RoboDK station: MPC Dental Surgery.rdk

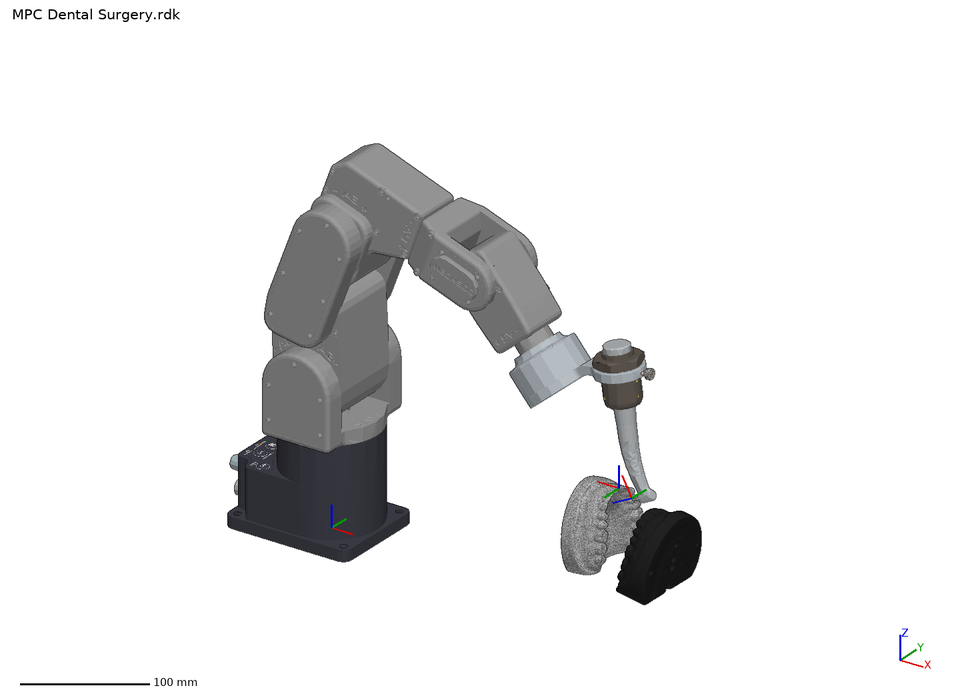
[picture v0: the station drawn from its stored meshes, robots at their saved joint values, targets as dots, program paths as lines]
Station MPC Dental Surgery (saved by RoboDK 5.3.5). Poses are relative to the parent item; angles as X-Y-Z fixed-axis rotations.
  - frame Mecademic Meca500 R3 Base at (0, 0, 0) mm
    - robot Mecademic Meca500 R3: 6 axes, payload 0.5 kg, reach 330 mm, repeatability 0.005 mm, weight 4.5 kg
        modified DH rows (alpha deg, a mm, theta deg, d mm): 0, 0, 0, 135; -90, 0, -90, 0; 0, 135, 0, 0; -90, 38, 0, 120; 90, 0, 0, 0; -90, 0, 180, 70
        joint limits [-175, -70, -135, -170, -115, -720] to [175, 90, 70, 170, 115, 720]; home [0, 0, 0, 0, 0, 0]; saved at [0, 10, 10, 0, 30, 0]
      - tool Assem, End Effector, V5_shortened v1, TCP at (0, 0, 0) mm, size 148.9 x 117.9 x 68.5 mm, geometry from Assem, End Effector, V5_shortened v1.step
      - frame Tool Center Point at (0, 0, 137) mm, rotated rx -180 ry 77 rz 180 deg
  - frame Patient Reference Frame at (200, 100, 50) mm, rotated rx 0 ry 0 rz 180 deg
    - object jaw at (-47, 0, -75) mm, rotated rx 10 ry 0 rz -90 deg, size 77.5 x 91.7 x 70.4 mm, geometry from jaw.step
